(* Logix 5000 project; controller Emulated_FlexFarm vendor 1 type 14 code 196 rev 36.11; software revision 36.00 *)

TASK MainTask (continuous, watchdog 500 ms) : MainProgram

MODULES
   Local : vendor 1 type 14 code 196 (5069 0, rev 36.11)
END_MODULES

VAR_GLOBAL   (* controller tags *)
   E3D_EC_TargetMax : DINT;   // Maximum EC value, Parameter set in E3D
   E3D_EC_TargetMin : DINT;   // Minimum EC value, Parameter set in E3D
   E3D_EC_Value : DINT;   // EC Value from E3D
   E3D_pH_TargetMax : DINT;   // Maximum pH value, Parameter set in E3D
   E3D_pH_TargetMin : DINT;   // Minimum pH value, Parameter set in E3D
   E3D_pH_Value : DINT;   // pH Value from E3D
   E3D_Water_TargetMax : DINT;   // Maximum water level value, Parameter set in E3D
   E3D_Water_TargetMin : DINT;   // Minimum water level value, Parameter set in E3D
   E3D_Water_Value : DINT;   // Water Level Value from E3D
   FreshWater_Pump : BOOL;   // Controls the activation of the Fresh Water pump in E3D
   Light_Control : BOOL := 1;   // Controls the activation of the Light in E3D
   Nutrient_Pump : BOOL;   // Controls the activation of the Nutrient pump in E3D
   pH_Pump : BOOL;   // Controls the activation of the pH pump in E3D
END_VAR

PROGRAM MainProgram   (* main routine MainRoutine *)
VAR
   steplogix : DINT := 1;
   TIMER : TIMER := (PRE := 18000, ACC := 12403, EN := 1, TT := 1);
   TIMER_1 : TIMER := (PRE := 6000);
END_VAR

ROUTINE Light_Control   (* ladder *)
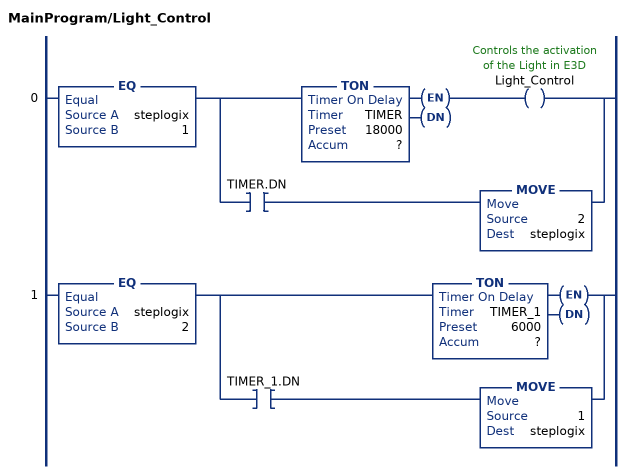
   0: EQ(steplogix,1)[TON(TIMER,?,?) OTE(Light_Control) ,XIC(TIMER.DN) MOVE(2,steplogix) ];
   1: EQ(steplogix,2)[TON(TIMER_1,?,?) ,XIC(TIMER_1.DN) MOVE(1,steplogix) ];
END_ROUTINE

ROUTINE MainRoutine   (* ladder *)
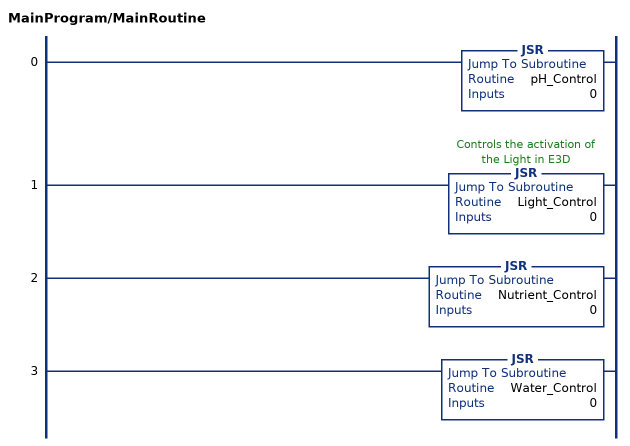
   0: JSR(pH_Control,0);
   1: JSR(Light_Control,0);
   2: JSR(Nutrient_Control,0);
   3: JSR(Water_Control,0);
END_ROUTINE

ROUTINE Nutrient_Control   (* ladder *)
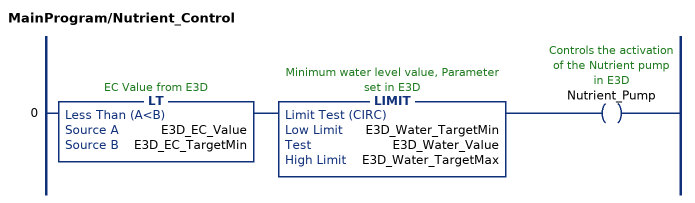
   0: LT(E3D_EC_Value,E3D_EC_TargetMin)LIMIT(E3D_Water_TargetMin,E3D_Water_Value,E3D_Water_TargetMax)OTE(Nutrient_Pump);
END_ROUTINE

ROUTINE pH_Control   (* ladder *)
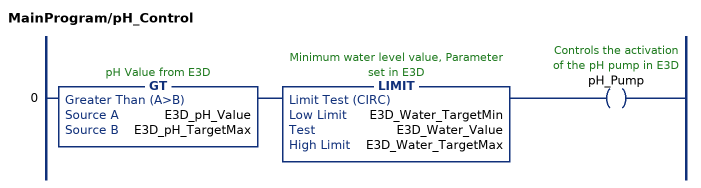
   0: GT(E3D_pH_Value,E3D_pH_TargetMax)LIMIT(E3D_Water_TargetMin,E3D_Water_Value,E3D_Water_TargetMax)OTE(pH_Pump);
END_ROUTINE

ROUTINE Water_Control   (* ladder *)
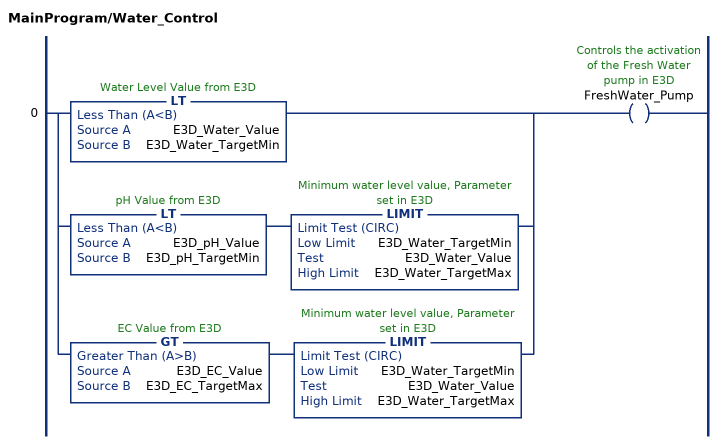
   0: [LT(E3D_Water_Value,E3D_Water_TargetMin) ,LT(E3D_pH_Value,E3D_pH_TargetMin) LIMIT(E3D_Water_TargetMin,E3D_Water_Value,E3D_Water_TargetMax) ,GT(E3D_EC_Value,E3D_EC_TargetMax) LIMIT(E3D_Water_TargetMin,E3D_Water_Value,E3D_Water_TargetMax) ]OTE(FreshWater_Pump);
END_ROUTINE
END_PROGRAM
